(* PLC project pumping, Dassault Systèmes ControlBuild 2024x *)
(* stored: creationDateTime 2023-10-03T11:13:42-01:00 *)

PROGRAM bottling_line.pumping
  VAR_INPUT
    fillingValve : BOOL := false;
    emptyingValve : BOOL := false;
    extractionPump : BOOL := false;
  END_VAR
  VAR_INPUT
    acknowledgePB : BOOL := false;
  END_VAR
  VAR_INPUT
    autoMode : BOOL := false;
    manualMode : BOOL := false;
  END_VAR
  VAR_OUTPUT
    lowLevel : BOOL := false;
    highLevel : BOOL := false;
  END_VAR
  VAR_OUTPUT
    pumpingFlow : REAL := 0.0;
    level : REAL := 0.0;
  END_VAR

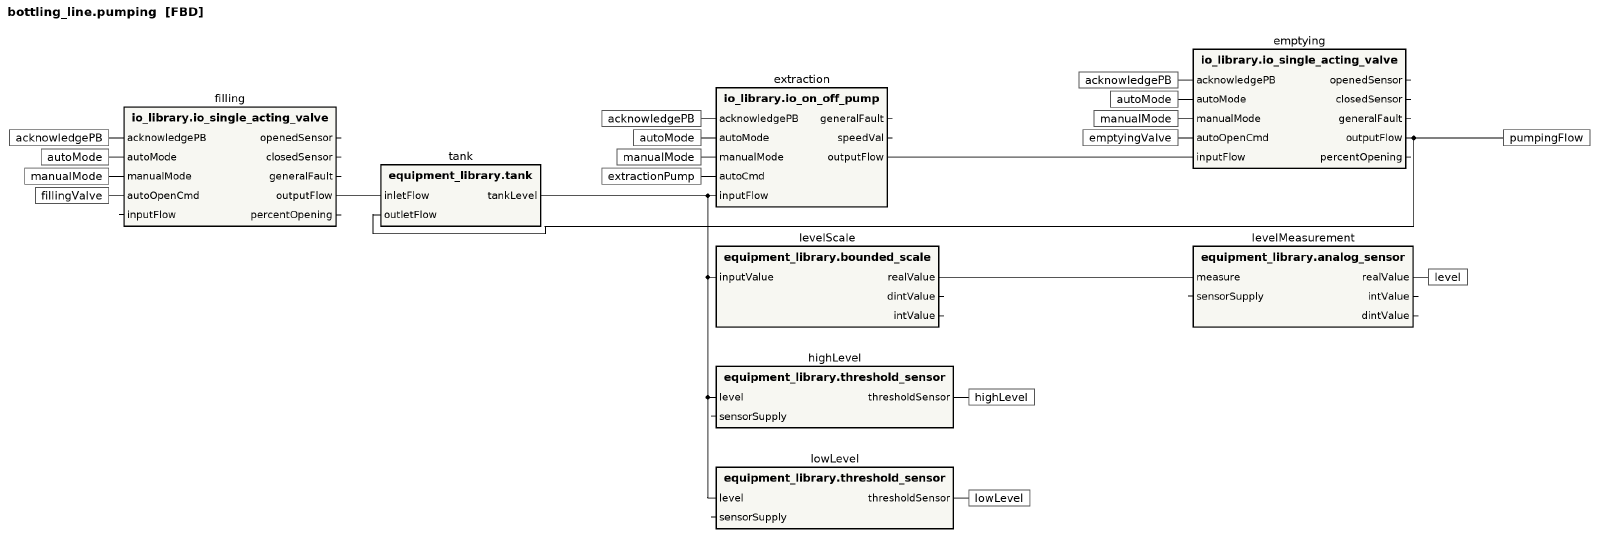
(* FBD diagram, written out as Structured Text *)
filling(acknowledgePB := acknowledgePB, autoMode := autoMode, manualMode := manualMode, autoOpenCmd := fillingValve);
extraction(acknowledgePB := acknowledgePB, autoMode := autoMode, manualMode := manualMode, autoCmd := extractionPump, inputFlow := tank.tankLevel);
emptying(acknowledgePB := acknowledgePB, autoMode := autoMode, manualMode := manualMode, autoOpenCmd := emptyingValve, inputFlow := extraction.outputFlow);
tank(inletFlow := filling.outputFlow, outletFlow := emptying.outputFlow);
levelScale(inputValue := tank.tankLevel);
levelMeasurement(measure := levelScale.realValue);
level := levelMeasurement.realValue;
highLevel(level := tank.tankLevel);
highLevel := highLevel.thresholdSensor;
lowLevel(level := tank.tankLevel);
lowLevel := lowLevel.thresholdSensor;
pumpingFlow := emptying.outputFlow;
END_PROGRAM
